TYPE ST_LA_Parameter :
STRUCT
	Temp_Kuehlwasser_Max	: REAL ;
	Temp_Kuehlwasser_Min	: REAL ;

	AutoQuittierung			: BOOL ;


	Abluefter_Druck_Sollwert 		: REAL;


	Ausschaltverz_Anlage_nach_Taster: REAL;

	Betriebsart_Anlage_RM			: REAL;
	Betriebsartenschalter_Anlage 	: REAL;

	Freie_Nachtkuehlung_AT_Grenzwert		: REAL;
	Freie_Nachtkuehlung_Diff_AT_zu_RT_Grenzwert : REAL;
	Freie_Nachtkuehlung_Nacht_Raumsollwert 	: REAL;

	Seminarraum_CO2_Sollwert_bei_Lueftungsbetrieb : REAL;
	Seminarraum_Grenzwert_CO2_Lueftung_Aus 	: REAL;
	Seminarraum_Grenzwert_CO2_Lueftung_Ein 	: REAL;

	Sollwertschiebung_Anlage_Max_Sollwert 	: REAL;
	Sollwertschiebung_Anlage_Min_Sollwert 	: REAL;
	Sollwertschiebung_Anlage_Max_AT_Sollwert: REAL;
	Sollwertschiebung_Anlage_Min_AT_Sollwert: REAL;

	Zuluefter_Drucksollwert 		: REAL;

END_STRUCT
END_TYPE

(* stored: Version 1.1.0.1, ProductVersion 3.1.4024.9
   DUT ST_LA_Parameter: Id {e816e84a-4bb0-44cb-ae15-60ada7290920} *)
